(* IEC 61131-3 sources: std_i2980_v2.06_cp053/Source/IMM/ieccontrol/OperationMode1 (part 3) *)

(* ---- ABProduction.pu ---- *)
(*
@h    ! WARNING !
@h    The Kemro K2 system (including software) only meets category B according to EN 954-1,
@h    thus it is not intended for usage in safety-relevant control applications in the field
@h    of personal safety (e.g. emergency stop).
@h    To implement potentially necessary safety-relevant control tasks, always use additional
@h    external safety devices that are intended for the particular purpose, and meet the necessary
@h    functional safety.
@h    For further information see EN 954-1 (EN ISO 13849-1) and/or the K2-x00 user manual, chapter
@h    "CE conformity, directives and standards".

production statistic (good/bad part)
called by ABShotCounter in order to provide some additional production information
*)

IMPORT_OVER_LISTFILE
 cCompPDP
, cCompMotionProtectMold
, tsTraceLevel
, tevPartCheck
, tnBadPartReason
, tsProduction
, RTC
, FBDebugTrace
, tevPartCheckData

END_IMPORT

ALGORITHM_BLOCK ABProduction #DUMMY_EDIT_BLOCK

SYSTEM_VAR
 sv_TraceLevel : tsTraceLevel;
 sv_bBadPart : BOOL;
 sv_iProdCounterAct : DINT;
 sv_iShotCounterRetain : UDINT (* shot counter retain (used for lubrication) *);
 sv_iCavities : DINT;
 sv_BadPartReason : tnBadPartReason;
 sv_Production : tsProduction;
 sv_dShotTimeAct : DATE_AND_TIME;
END_VAR

SYSTEM_OBJECT
 evPartCheck : tevPartCheck;
 EV_Task_7 : TASK;
 PU_Task_7 : TASK;
END_OBJECT

VAR
 miRejectsPerTime : DINT;
 fbRtc : RTC;
 mdStartTime : DT;
 fbDebugTrace : FBDebugTrace;
END_VAR

(*
@h    ! WARNING !
@h    The Kemro K2 system (including software) only meets category B according to EN 954-1,
@h    thus it is not intended for usage in safety-relevant control applications in the field
@h    of personal safety (e.g. emergency stop).
@h    To implement potentially necessary safety-relevant control tasks, always use additional
@h    external safety devices that are intended for the particular purpose, and meet the necessary
@h    functional safety.
@h    For further information see EN 954-1 (EN ISO 13849-1) and/or the K2-x00 user manual, chapter
@h    "CE conformity, directives and standards".

reacts on partcheck events with bBadPart == TRUE,
sets sv_bBadPart and sv_BadPartReason
*)

EVENT_ALGORITHM evaPartCheck ON EV_Task_7 WITH evPartCheck

VAR_INPUT
 partCheckData : tevPartCheckData;
END_VAR

VAR
 s : STRING(255);
END_VAR
#BEGIN_EDIT_BLOCK
(**************************************** WARNING ********************************************
 *** The KEBA Kemro K2 System including software is not intended for safety control tasks! ***
 ***                       For further information see Comment tab!                        ***
 *********************************************************************************************)

IF sv_TraceLevel.bApplication THEN
    s := CONCAT('part check event recieved: device ',
                DINT_TO_STRING(partCheckData.DeviceID.CompId),
                '/',
                DINT_TO_STRING(partCheckData.DeviceID.IndexId),
                ' bad ',
                BOOL_TO_STRING(partCheckData.bBadPart),
                ' reject',
                BOOL_TO_STRING(partCheckData.bReject)
            );
    fbDebugTrace(sText := s);
END_IF;

IF partCheckData.bBadPart THEN
    sv_bBadPart := TRUE;

    // set bad part reason
    IF sv_BadPartReason = nReason_GoodPart THEN
       CASE (partCheckData.DeviceID.CompId) OF
            cCompPDP:
                 sv_BadPartReason := nReason_PDS;

            cCompMotionProtectMold:
                 sv_BadPartReason := nReason_MoldProtection;
       ELSE
             sv_BadPartReason := nReason_Unknown;
       END_CASE;
    END_IF;

END_IF;

;#END_EDIT_BLOCK END_ALGORITHM

(*
@h    ! WARNING !
@h    The Kemro K2 system (including software) only meets category B according to EN 954-1,
@h    thus it is not intended for usage in safety-relevant control applications in the field
@h    of personal safety (e.g. emergency stop).
@h    To implement potentially necessary safety-relevant control tasks, always use additional
@h    external safety devices that are intended for the particular purpose, and meet the necessary
@h    functional safety.
@h    For further information see EN 954-1 (EN ISO 13849-1) and/or the K2-x00 user manual, chapter
@h    "CE conformity, directives and standards".

called by ABShotCounter before shotcounter is increased, so sv_Production vars that can be recorded
by PDP are written before sampled by PDP
*)

ALGORITHM aNewCycle

#BEGIN_EDIT_BLOCK
(**************************************** WARNING ********************************************
 *** The KEBA Kemro K2 System including software is not intended for safety control tasks! ***
 ***                       For further information see Comment tab!                        ***
 *********************************************************************************************)

// end of actual cycle, calc some production data

fbRtc();
sv_dShotTimeAct := fbRtc.CDT;

IF ((fbRtc.CDT - mdStartTime) >= LINT_TO_TIME(DINT_TO_LINT(sv_Production.iRejectTimeSpan * 60 * 1000) * 1000)) THEN
    mdStartTime := fbRtc.CDT;
    sv_Production.iRejectsPerTime := miRejectsPerTime;
    miRejectsPerTime := 0;
END_IF;

IF sv_bBadPart THEN
    sv_Production.iRejectCounter := sv_Production.iRejectCounter + sv_iCavities;
    miRejectsPerTime := miRejectsPerTime + sv_iCavities;
    sv_Production.iRejectsInSeries := sv_Production.iRejectsInSeries + 1;
ELSE
    sv_Production.iRejectsInSeries := 0;
END_IF;

IF sv_Production.iRejectCounter > 0 THEN
    sv_Production.iGoodPartsPerReject := (sv_iProdCounterAct - sv_Production.iRejectCounter) / sv_Production.iRejectCounter;
END_IF;

;#END_EDIT_BLOCK END_ALGORITHM

(*
@h    ! WARNING !
@h    The Kemro K2 system (including software) only meets category B according to EN 954-1,
@h    thus it is not intended for usage in safety-relevant control applications in the field
@h    of personal safety (e.g. emergency stop).
@h    To implement potentially necessary safety-relevant control tasks, always use additional
@h    external safety devices that are intended for the particular purpose, and meet the necessary
@h    functional safety.
@h    For further information see EN 954-1 (EN ISO 13849-1) and/or the K2-x00 user manual, chapter
@h    "CE conformity, directives and standards".

called by ABShotCounter when shotcounter is reset
to clear all production statistics variables also
*)

ALGORITHM aResetData

#BEGIN_EDIT_BLOCK
(**************************************** WARNING ********************************************
 *** The KEBA Kemro K2 System including software is not intended for safety control tasks! ***
 ***                       For further information see Comment tab!                        ***
 *********************************************************************************************)

sv_Production.iRejectCounter := 0;
sv_Production.iRejectsPerTime := 0;
sv_Production.iGoodPartsPerReject := 2147483647;
sv_Production.iRejectsInSeries := 0;

miRejectsPerTime := 0;
fbRtc();
mdStartTime := fbRtc.CDT;

;#END_EDIT_BLOCK END_ALGORITHM

(*
@h    ! WARNING !
@h    The Kemro K2 system (including software) only meets category B according to EN 954-1,
@h    thus it is not intended for usage in safety-relevant control applications in the field
@h    of personal safety (e.g. emergency stop).
@h    To implement potentially necessary safety-relevant control tasks, always use additional
@h    external safety devices that are intended for the particular purpose, and meet the necessary
@h    functional safety.
@h    For further information see EN 954-1 (EN ISO 13849-1) and/or the K2-x00 user manual, chapter
@h    "CE conformity, directives and standards".

called when new cycle starts (shotcounter has just been increased) but lower prio than PDP recording
so SVs to be recorded by PDP are sampled before reset
*)

POSTUPDATE_ALGORITHM pNewCycle ON PU_Task_7 WITH sv_iShotCounterRetain

#BEGIN_EDIT_BLOCK
(**************************************** WARNING ********************************************
 *** The KEBA Kemro K2 System including software is not intended for safety control tasks! ***
 ***                       For further information see Comment tab!                        ***
 *********************************************************************************************)

//reset bad part
// ATTENTION: lower prio than PDP MS Task so PDP has recorded these SVs before reset!

sv_bBadPart := FALSE;
sv_BadPartReason := nReason_GoodPart;

;#END_EDIT_BLOCK END_ALGORITHM

END_ALGORITHM_BLOCK

#END_OF_IEC_PART

@Puma @IecEditor 6 103 @Pou 25
@@@BEG_Comment@@@
@h    ! WARNING !
@h    The Kemro K2 system (including software) only meets category B according to EN 954-1,
@h    thus it is not intended for usage in safety-relevant control applications in the field
@h    of personal safety (e.g. emergency stop).
@h    To implement potentially necessary safety-relevant control tasks, always use additional
@h    external safety devices that are intended for the particular purpose, and meet the necessary
@h    functional safety.
@h    For further information see EN 954-1 (EN ISO 13849-1) and/or the K2-x00 user manual, chapter
@h    "CE conformity, directives and standards".

production statistic (good/bad part)
called by ABShotCounter in order to provide some additional production information
@@@END_Comment@@@

@BEG_Contents

@BEG_Func
@RT(17)FuncTreeContainer
0
@END_Func

@BEG_Const
@RT(18)ConstTreeContainer
2
@Var @RT(8)cCompPDP @RT(0) @T @F @DT @RT(4)DINT @RT(0) @T @T @BASIC 0 @F
@F @F
@T
@BEG_Attrib
0 @RT(3)119 @RT(30)Component Process Data Package
@END_Attrib
1 1 @F @F @F @F

@Var @RT(22)cCompMotionProtectMold @RT(0) @T @F @DT @RT(4)DINT @RT(0) @T @T @BASIC 0 @F
@F @F
@T
@BEG_Attrib
0 @RT(3)130 @RT(29)Component Motion Protect Mold
@END_Attrib
1 1 @F @F @F @F

@END_Const

@BEG_Export

@BEG_Kind
@ALGORITHM_BLOCK @RT(12)ABProduction @STRUCTURED_TEXT
@RT(0) @RT(0) @RT(0)
@END_Kind

@BEG_Dcl
@RT(16)DclTreeContainer
15
@Var @RT(13)sv_TraceLevel @RT(0) @T @T @DERIVED 0 @T @T @DT @RT(12)tsTraceLevel @RT(0) @T @T @UNKNOWN 0 @F
@F @F
@T
@BEG_Attrib
3 @RT(0) @RT(0) @RT(0)
@END_Attrib
1 8 @F @F @F @F

@Var @RT(11)evPartCheck @RT(0) @T @T @DERIVED 0 @T @T @DT @RT(12)tevPartCheck @RT(0) @T @T @UNKNOWN 0 @F
@F @F
@T
@BEG_Attrib
3 @RT(0) @RT(0) @RT(0)
@END_Attrib
1 7 @F @F @F @F

@Var @RT(9)EV_Task_7 @RT(0) @T @T @RENAMED 0 @T @T @DT @RT(4)TASK @RT(0) @T @T @BASIC 0 @F
@F @F
@T
@BEG_Attrib
3 @RT(0) @RT(0) @RT(0)
@END_Attrib
1 7 @F @F @F @F

@Var @RT(11)sv_bBadPart @RT(0) @T @F @DT @RT(4)BOOL @RT(0) @T @T @BASIC 0 @F
@F @F
@T
@BEG_Attrib
3 @RT(0) @RT(0) @RT(0)
@END_Attrib
1 8 @F @F @F @F

@Var @RT(18)sv_iProdCounterAct @RT(0) @T @F @DT @RT(4)DINT @RT(0) @T @T @BASIC 0 @F
@F @F
@T
@BEG_Attrib
3 @RT(0) @RT(0) @RT(0)
@END_Attrib
1 8 @F @F @F @F

@Var @RT(21)sv_iShotCounterRetain @RT(0) @T @F @DT @RT(5)UDINT @RT(0) @T @T @BASIC 0 @F
@F @F
@T
@BEG_Attrib
3 @RT(0) @RT(42)shot counter retain (used for lubrication) @RT(0)
@END_Attrib
1 8 @F @F @F @F

@Var @RT(12)sv_iCavities @RT(0) @T @F @DT @RT(4)DINT @RT(0) @T @T @BASIC 0 @F
@F @F
@T
@BEG_Attrib
3 @RT(0) @RT(0) @RT(0)
@END_Attrib
1 8 @F @F @F @F

@Var @RT(16)sv_BadPartReason @RT(0) @T @T @DERIVED 0 @T @T @DT @RT(15)tnBadPartReason @RT(0) @T @T @UNKNOWN 0 @F
@F @F
@T
@BEG_Attrib
3 @RT(0) @RT(0) @RT(0)
@END_Attrib
1 8 @F @F @F @F

@Var @RT(13)sv_Production @RT(0) @T @T @DERIVED 0 @T @T @DT @RT(12)tsProduction @RT(0) @T @T @UNKNOWN 0 @F
@F @F
@T
@BEG_Attrib
3 @RT(0) @RT(0) @RT(0)
@END_Attrib
1 8 @F @F @F @F

@Var @RT(16)miRejectsPerTime @RT(0) @T @F @DT @RT(4)DINT @RT(0) @T @T @BASIC 0 @F
@F @F
@T
@BEG_Attrib
3 @RT(0) @RT(0) @RT(0)
@END_Attrib
1 0 @F @F @F @F

@Var @RT(5)fbRtc @RT(0) @T @T @DERIVED 0 @T @T @DT @RT(3)RTC @RT(0) @T @T @UNKNOWN 0 @F
@F @F
@T
@BEG_Attrib
3 @RT(0) @RT(0) @RT(0)
@END_Attrib
1 0 @F @F @F @F

@Var @RT(15)sv_dShotTimeAct @RT(0) @T @F @DT @RT(13)DATE_AND_TIME @RT(0) @T @T @BASIC 0 @F
@F @F
@T
@BEG_Attrib
3 @RT(0) @RT(0) @RT(0)
@END_Attrib
1 8 @F @F @F @F

@Var @RT(11)mdStartTime @RT(0) @T @F @DT @RT(2)DT @RT(0) @T @T @BASIC 0 @F
@F @F
@T
@BEG_Attrib
3 @RT(0) @RT(0) @RT(0)
@END_Attrib
1 0 @F @F @F @F

@Var @RT(9)PU_Task_7 @RT(0) @T @T @RENAMED 0 @T @T @DT @RT(4)TASK @RT(0) @T @T @BASIC 0 @F
@F @F
@T
@BEG_Attrib
3 @RT(0) @RT(0) @RT(0)
@END_Attrib
1 7 @F @F @F @F

@Var @RT(12)fbDebugTrace @RT(0) @T @T @DERIVED 0 @T @T @DT @RT(12)FBDebugTrace @RT(0) @T @T @UNKNOWN 0 @F
@F @F
@T
@BEG_Attrib
3 @RT(0) @RT(0) @RT(0)
@END_Attrib
1 0 @F @F @F @F

@END_Dcl

@END_Export

@BEG_Body

4

@BEG_Export

@BEG_Algo
@EVENT_ALGORITHM @RT(12)evaPartCheck @STRUCTURED_TEXT
@RT(0) @RT(11)evPartCheck @RT(9)EV_Task_7 @F @F
@END_Algo

@BEG_Dcl
@RT(16)DclTreeContainer
2
@Var @RT(13)partCheckData @RT(0) @T @T @DERIVED 0 @T @T @DT @RT(16)tevPartCheckData @RT(0) @T @T @UNKNOWN 0 @F
@F @F
@T
@BEG_Attrib
3 @RT(0) @RT(0) @RT(0)
@END_Attrib
1 1 @F @F @F @F

@Var @RT(1)s @RT(0) @T @F @DT @RT(11)STRING(255) @RT(0) @T @T @STRING 0 @F @RT(3)255 @F
@F @F
@T
@BEG_Attrib
3 @RT(0) @RT(0) @RT(0)
@END_Attrib
1 0 @F @F @F @F

@END_Dcl

@END_Export

@BEG_Export

@BEG_Algo
@ALGORITHM @RT(9)aNewCycle @STRUCTURED_TEXT
@RT(0) @RT(0) @RT(0) @F @F
@END_Algo

@BEG_Dcl
@RT(16)DclTreeContainer
0
@END_Dcl

@END_Export

@BEG_Export

@BEG_Algo
@ALGORITHM @RT(10)aResetData @STRUCTURED_TEXT
@RT(0) @RT(0) @RT(0) @F @F
@END_Algo

@BEG_Dcl
@RT(16)DclTreeContainer
0
@END_Dcl

@END_Export

@BEG_Export

@BEG_Algo
@POSTUPDATE_ALGORITHM @RT(9)pNewCycle @STRUCTURED_TEXT
@RT(0) @RT(21)sv_iShotCounterRetain @RT(9)PU_Task_7 @F @F
@END_Algo

@BEG_Dcl
@RT(16)DclTreeContainer
0
@END_Dcl

@END_Export

@BEG_Body
@TL(38)
(**************************************** WARNING ********************************************
 *** The KEBA Kemro K2 System including software is not intended for safety control tasks! ***
 ***                       For further information see Comment tab!                        ***
 *********************************************************************************************)

IF sv_TraceLevel.bApplication THEN
    s := CONCAT('part check event recieved: device ',
                DINT_TO_STRING(partCheckData.DeviceID.CompId),
                '/',
                DINT_TO_STRING(partCheckData.DeviceID.IndexId),
                ' bad ',
                BOOL_TO_STRING(partCheckData.bBadPart),
                ' reject',
                BOOL_TO_STRING(partCheckData.bReject)
            );
    fbDebugTrace(sText := s);
END_IF;

IF partCheckData.bBadPart THEN
    sv_bBadPart := TRUE;

    // set bad part reason
    IF sv_BadPartReason = nReason_GoodPart THEN
       CASE (partCheckData.DeviceID.CompId) OF
            cCompPDP:
                 sv_BadPartReason := nReason_PDS;

            cCompMotionProtectMold:
                 sv_BadPartReason := nReason_MoldProtection;
       ELSE
             sv_BadPartReason := nReason_Unknown;
       END_CASE;
    END_IF;

END_IF;

@END_Body

@@@BEG_Comment@@@
@TL(12)
@h    ! WARNING !
@h    The Kemro K2 system (including software) only meets category B according to EN 954-1,
@h    thus it is not intended for usage in safety-relevant control applications in the field
@h    of personal safety (e.g. emergency stop).
@h    To implement potentially necessary safety-relevant control tasks, always use additional
@h    external safety devices that are intended for the particular purpose, and meet the necessary
@h    functional safety.
@h    For further information see EN 954-1 (EN ISO 13849-1) and/or the K2-x00 user manual, chapter
@h    "CE conformity, directives and standards".

reacts on partcheck events with bBadPart == TRUE,
sets sv_bBadPart and sv_BadPartReason
@@@END_Comment@@@

@BEG_Body
@TL(30)
(**************************************** WARNING ********************************************
 *** The KEBA Kemro K2 System including software is not intended for safety control tasks! ***
 ***                       For further information see Comment tab!                        ***
 *********************************************************************************************)

// end of actual cycle, calc some production data

fbRtc();
sv_dShotTimeAct := fbRtc.CDT;

IF ((fbRtc.CDT - mdStartTime) >= LINT_TO_TIME(DINT_TO_LINT(sv_Production.iRejectTimeSpan * 60 * 1000) * 1000)) THEN
    mdStartTime := fbRtc.CDT;
    sv_Production.iRejectsPerTime := miRejectsPerTime;
    miRejectsPerTime := 0;
END_IF;

IF sv_bBadPart THEN
    sv_Production.iRejectCounter := sv_Production.iRejectCounter + sv_iCavities;
    miRejectsPerTime := miRejectsPerTime + sv_iCavities;
    sv_Production.iRejectsInSeries := sv_Production.iRejectsInSeries + 1;
ELSE
    sv_Production.iRejectsInSeries := 0;
END_IF;

IF sv_Production.iRejectCounter > 0 THEN
    sv_Production.iGoodPartsPerReject := (sv_iProdCounterAct - sv_Production.iRejectCounter) / sv_Production.iRejectCounter;
END_IF;

@END_Body

@@@BEG_Comment@@@
@TL(12)
@h    ! WARNING !
@h    The Kemro K2 system (including software) only meets category B according to EN 954-1,
@h    thus it is not intended for usage in safety-relevant control applications in the field
@h    of personal safety (e.g. emergency stop).
@h    To implement potentially necessary safety-relevant control tasks, always use additional
@h    external safety devices that are intended for the particular purpose, and meet the necessary
@h    functional safety.
@h    For further information see EN 954-1 (EN ISO 13849-1) and/or the K2-x00 user manual, chapter
@h    "CE conformity, directives and standards".

called by ABShotCounter before shotcounter is increased, so sv_Production vars that can be recorded
by PDP are written before sampled by PDP
@@@END_Comment@@@

@BEG_Body
@TL(14)
(**************************************** WARNING ********************************************
 *** The KEBA Kemro K2 System including software is not intended for safety control tasks! ***
 ***                       For further information see Comment tab!                        ***
 *********************************************************************************************)

sv_Production.iRejectCounter := 0;
sv_Production.iRejectsPerTime := 0;
sv_Production.iGoodPartsPerReject := 2147483647;
sv_Production.iRejectsInSeries := 0;

miRejectsPerTime := 0;
fbRtc();
mdStartTime := fbRtc.CDT;

@END_Body

@@@BEG_Comment@@@
@TL(12)
@h    ! WARNING !
@h    The Kemro K2 system (including software) only meets category B according to EN 954-1,
@h    thus it is not intended for usage in safety-relevant control applications in the field
@h    of personal safety (e.g. emergency stop).
@h    To implement potentially necessary safety-relevant control tasks, always use additional
@h    external safety devices that are intended for the particular purpose, and meet the necessary
@h    functional safety.
@h    For further information see EN 954-1 (EN ISO 13849-1) and/or the K2-x00 user manual, chapter
@h    "CE conformity, directives and standards".

called by ABShotCounter when shotcounter is reset
to clear all production statistics variables also
@@@END_Comment@@@

@BEG_Body
@TL(12)
(**************************************** WARNING ********************************************
 *** The KEBA Kemro K2 System including software is not intended for safety control tasks! ***
 ***                       For further information see Comment tab!                        ***
 *********************************************************************************************)

//reset bad part
// ATTENTION: lower prio than PDP MS Task so PDP has recorded these SVs before reset!

sv_bBadPart := FALSE;
sv_BadPartReason := nReason_GoodPart;

@END_Body

@@@BEG_Comment@@@
@TL(12)
@h    ! WARNING !
@h    The Kemro K2 system (including software) only meets category B according to EN 954-1,
@h    thus it is not intended for usage in safety-relevant control applications in the field
@h    of personal safety (e.g. emergency stop).
@h    To implement potentially necessary safety-relevant control tasks, always use additional
@h    external safety devices that are intended for the particular purpose, and meet the necessary
@h    functional safety.
@h    For further information see EN 954-1 (EN ISO 13849-1) and/or the K2-x00 user manual, chapter
@h    "CE conformity, directives and standards".

called when new cycle starts (shotcounter has just been increased) but lower prio than PDP recording
so SVs to be recorded by PDP are sampled before reset
@@@END_Comment@@@
@END_Body

@END_Contents

(* ---- ABSequenceInterruption.pu ---- *)
(*
@h    ! WARNING !
@h    The Kemro K2 system (including software) only meets category B according to EN 954-1,
@h    thus it is not intended for usage in safety-relevant control applications in the field
@h    of personal safety (e.g. emergency stop).
@h    To implement potentially necessary safety-relevant control tasks, always use additional
@h    external safety devices that are intended for the particular purpose, and meet the necessary
@h    functional safety.
@h    For further information see EN 954-1 (EN ISO 13849-1) and/or the K2-x00 user manual, chapter
@h    "CE conformity, directives and standards".

This AB is responsible for setting / resetting the flag for sequence interruption (sv_bSequenceInterruption).
A sequence interruption can be triggered by any function unit. Therefore and according event (evSequenceInterrupt)
must be sent.
This block can also handle a seperate digital input (di_SequenceInterruption) which can trigger an interrupt.
Interrupt events (or the according digital input) are ignored in manual and setup mode.

During sequence is interrupted, the led for halfautocycle or fullautocycle is set to "flashing"

*)

IMPORT_OVER_LISTFILE
 tnOperationMode
, tevSequenceInterrupt
, tsActiveMovements
, tevSequInterruptData

END_IMPORT

ALGORITHM_BLOCK ABSequenceInterruption #DUMMY_EDIT_BLOCK

SYSTEM_VAR
 di_SequenceInterruption : BOOL;
 sv_bSequenceInterruption : BOOL (* TRUE: sequence is interrupted *);
 sv_bLedHalfAutomatic_ledAttr : BYTE (* Panel LED half automatic *);
 sv_bLedFullAutomatic_ledAttr : BYTE (* Panel LED full automatic *);
 sv_bHMILedHalfAutomatic_ledAttr : BYTE (* Panel LED half automatic *);
 sv_bHMILedFullAutomatic_ledAttr : BYTE (* Panel LED full automatic *);
 sv_OperationMode : tnOperationMode;
 sv_ActiveMovements : tsActiveMovements;
END_VAR

SYSTEM_OBJECT
 PU_Task_7 : TASK;
 EV_Task_7 : TASK;
 evSequenceInterrupt : tevSequenceInterrupt;
 TaskMid : TASK;
END_OBJECT

VAR
 mbLedHalfAutomaticAttrLinked : BOOL;
 mbLedFullAutomaticAttrLinked : BOOL;
 mbResetInterrupt : BOOL;
END_VAR

POSTUPDATE_ALGORITHM pDISequenceInterrupt ON PU_Task_7 WITH di_SequenceInterruption

VAR
 evSequenceInterruptData : tevSequInterruptData;
END_VAR
#BEGIN_EDIT_BLOCK
(**************************************** WARNING ********************************************
 *** The KEBA Kemro K2 System including software is not intended for safety control tasks! ***
 ***                       For further information see Comment tab!                        ***
 *********************************************************************************************)

IF di_SequenceInterruption THEN
   IF sv_bSequenceInterruption THEN
      evSequenceInterruptData.SequenceInterrupt := nSequenceContinue;
   ELSE
      evSequenceInterruptData.SequenceInterrupt := nSequenceInterrupt;
   END_IF;

   SET_EVENT(evSequenceInterrupt, evSequenceInterruptData);
END_IF;

;#END_EDIT_BLOCK END_ALGORITHM

EVENT_ALGORITHM evaSequenceInterrupt ON EV_Task_7 WITH evSequenceInterrupt

VAR_INPUT
 evSequInterruptData : tevSequInterruptData;
END_VAR
#BEGIN_EDIT_BLOCK
(**************************************** WARNING ********************************************
 *** The KEBA Kemro K2 System including software is not intended for safety control tasks! ***
 ***                       For further information see Comment tab!                        ***
 *********************************************************************************************)

IF (sv_OperationMode = nSetup) OR (sv_OperationMode = nManual) THEN
   RETURN;
END_IF;

IF evSequInterruptData.SequenceInterrupt = nSequenceInterrupt THEN
   sv_bSequenceInterruption := TRUE;
   mbResetInterrupt := FALSE;

   //set led attribute to "flashing" during sequence interrupt
   sv_bLedHalfAutomatic_ledAttr := 16#3;
   sv_bLedFullAutomatic_ledAttr := 16#3;

   sv_bHMILedHalfAutomatic_ledAttr := sv_bLedHalfAutomatic_ledAttr;
   sv_bHMILedFullAutomatic_ledAttr := sv_bLedFullAutomatic_ledAttr;

   START_PROCESS_ALGORITHM(paSequenceInterrupted);
ELSE
   mbResetInterrupt := TRUE;
END_IF;

;#END_EDIT_BLOCK END_ALGORITHM

PROCESS_ALGORITHM paSequenceInterrupted ON TaskMid

(* IecGraph-Code *)

(* init step *)
INITIAL_STEP S_Init:
Action9 (P);
END_STEP

ACTION Action9: #BEGIN_EDIT_BLOCK

mbLedHalfAutomaticAttrLinked := IS_LINKED(sv_bLedHalfAutomatic_ledAttr);
mbLedFullAutomaticAttrLinked := IS_LINKED(sv_bLedFullAutomatic_ledAttr);

;#END_EDIT_BLOCK END_ACTION (*Action9*)

(* steps *)
STEP S_Interrupted:
END_STEP

STEP S_WaitNoMove:
END_STEP

STEP S_Stop:
AReset (P);
AStop (P);
END_STEP

ACTION AReset: #BEGIN_EDIT_BLOCK
sv_bSequenceInterruption := FALSE;
//set led attribute to "not flashing"
sv_bHMILedHalfAutomatic_ledAttr := 16#1;
sv_bHMILedFullAutomatic_ledAttr := 16#1;

IF mbLedHalfAutomaticAttrLinked THEN
   sv_bLedHalfAutomatic_ledAttr := sv_bHMILedHalfAutomatic_ledAttr;
END_IF;

IF mbLedFullAutomaticAttrLinked THEN
   sv_bLedFullAutomatic_ledAttr := sv_bHMILedFullAutomatic_ledAttr;
END_IF;

;#END_EDIT_BLOCK END_ACTION (*AReset*)
ACTION AStop: #BEGIN_EDIT_BLOCK
STOP_PROCESS_ALGORITHM();

;#END_EDIT_BLOCK END_ACTION (*AStop*)

(* transitions *)
GO_ON_TRANSITION Trans1 (* Trans1 *) FROM S_Init TO S_Interrupted :=  #BEGIN_EDIT_BLOCK
TRUE
;#END_EDIT_BLOCK
END_TRANSITION

GO_ON_TRANSITION TResetInterrupt (* Trans2 *) FROM S_Interrupted TO S_WaitNoMove :=  #BEGIN_EDIT_BLOCK
mbResetInterrupt
;#END_EDIT_BLOCK
END_TRANSITION

GO_ON_TRANSITION TNoMovementActive (* Trans4 *) FROM S_WaitNoMove TO S_Stop :=  #BEGIN_EDIT_BLOCK
sv_ActiveMovements.iNumberOfActiveMovements = 0
;#END_EDIT_BLOCK
END_TRANSITION

GO_ON_TRANSITION TOpModeChanged (* Trans8 *) FROM S_Interrupted TO S_Stop :=  #BEGIN_EDIT_BLOCK
sv_OperationMode < nHalfAutomatic
;#END_EDIT_BLOCK
END_TRANSITION

TRANSITION Trans3 (* Trans3 *) FROM S_Stop TO S_Interrupted :=  #BEGIN_EDIT_BLOCK
TRUE
;#END_EDIT_BLOCK
END_TRANSITION

(* end IecGraph-Code *)
(* sfc-code *)

(* stand alone actions *)
// ACTION Action9: #BEGIN_EDIT_BLOCK

// ;#END_EDIT_BLOCK END_ACTION (*Action9*)
(* end sfc-code *)

END_ALGORITHM

END_ALGORITHM_BLOCK

#END_OF_IEC_PART

@Puma @IecEditor 6 131 @Pou 25
@@@BEG_Comment@@@
@h    ! WARNING !
@h    The Kemro K2 system (including software) only meets category B according to EN 954-1,
@h    thus it is not intended for usage in safety-relevant control applications in the field
@h    of personal safety (e.g. emergency stop).
@h    To implement potentially necessary safety-relevant control tasks, always use additional
@h    external safety devices that are intended for the particular purpose, and meet the necessary
@h    functional safety.
@h    For further information see EN 954-1 (EN ISO 13849-1) and/or the K2-x00 user manual, chapter
@h    "CE conformity, directives and standards".

This AB is responsible for setting / resetting the flag for sequence interruption (sv_bSequenceInterruption).
A sequence interruption can be triggered by any function unit. Therefore and according event (evSequenceInterrupt)
must be sent.
This block can also handle a seperate digital input (di_SequenceInterruption) which can trigger an interrupt.
Interrupt events (or the according digital input) are ignored in manual and setup mode.

During sequence is interrupted, the led for halfautocycle or fullautocycle is set to "flashing"

@@@END_Comment@@@

@BEG_Contents

@BEG_Func
@RT(17)FuncTreeContainer
0
@END_Func

@BEG_Const
@RT(18)ConstTreeContainer
0
@END_Const

@BEG_Export

@BEG_Kind
@ALGORITHM_BLOCK @RT(22)ABSequenceInterruption @STRUCTURED_TEXT
@RT(0) @RT(0) @RT(0)
@END_Kind

@BEG_Dcl
@RT(16)DclTreeContainer
15
@Var @RT(23)di_SequenceInterruption @RT(0) @T @F @DT @RT(4)BOOL @RT(0) @T @T @BASIC 0 @F
@F @F
@T
@BEG_Attrib
3 @RT(0) @RT(0) @RT(0)
@END_Attrib
1 8 @F @F @F @F

@Var @RT(9)PU_Task_7 @RT(0) @T @T @RENAMED 0 @T @T @DT @RT(4)TASK @RT(0) @T @T @BASIC 0 @F
@F @F
@T
@BEG_Attrib
3 @RT(0) @RT(0) @RT(0)
@END_Attrib
1 7 @F @F @F @F

@Var @RT(24)sv_bSequenceInterruption @RT(0) @T @F @DT @RT(4)BOOL @RT(0) @T @T @BASIC 0 @F
@F @F
@T
@BEG_Attrib
3 @RT(0) @RT(29)TRUE: sequence is interrupted @RT(0)
@END_Attrib
1 8 @F @F @F @F

@Var @RT(28)sv_bLedHalfAutomatic_ledAttr @RT(0) @T @F @DT @RT(4)BYTE @RT(0) @T @T @BASIC 0 @F
@F @F
@T
@BEG_Attrib
3 @RT(0) @RT(24)Panel LED half automatic @RT(0)
@END_Attrib
1 8 @F @F @F @F

@Var @RT(28)sv_bLedFullAutomatic_ledAttr @RT(0) @T @F @DT @RT(4)BYTE @RT(0) @T @T @BASIC 0 @F
@F @F
@T
@BEG_Attrib
3 @RT(0) @RT(24)Panel LED full automatic @RT(0)
@END_Attrib
1 8 @F @F @F @F

@Var @RT(31)sv_bHMILedHalfAutomatic_ledAttr @RT(0) @T @F @DT @RT(4)BYTE @RT(0) @T @T @BASIC 0 @F
@F @F
@T
@BEG_Attrib
3 @RT(0) @RT(24)Panel LED half automatic @RT(0)
@END_Attrib
1 8 @F @F @F @F

@Var @RT(31)sv_bHMILedFullAutomatic_ledAttr @RT(0) @T @F @DT @RT(4)BYTE @RT(0) @T @T @BASIC 0 @F
@F @F
@T
@BEG_Attrib
3 @RT(0) @RT(24)Panel LED full automatic @RT(0)
@END_Attrib
1 8 @F @F @F @F

@Var @RT(16)sv_OperationMode @RT(0) @T @T @DERIVED 0 @T @T @DT @RT(15)tnOperationMode @RT(0) @T @T @UNKNOWN 0 @F
@F @F
@T
@BEG_Attrib
3 @RT(0) @RT(0) @RT(0)
@END_Attrib
1 8 @F @F @F @F

@Var @RT(9)EV_Task_7 @RT(0) @T @T @RENAMED 0 @T @T @DT @RT(4)TASK @RT(0) @T @T @BASIC 0 @F
@F @F
@T
@BEG_Attrib
3 @RT(0) @RT(0) @RT(0)
@END_Attrib
1 7 @F @F @F @F

@Var @RT(19)evSequenceInterrupt @RT(0) @T @T @DERIVED 0 @T @T @DT @RT(20)tevSequenceInterrupt @RT(0) @T @T @UNKNOWN 0 @F
@F @F
@T
@BEG_Attrib
3 @RT(0) @RT(0) @RT(0)
@END_Attrib
1 7 @F @F @F @F

@Var @RT(7)TaskMid @RT(0) @T @T @RENAMED 0 @T @T @DT @RT(4)TASK @RT(0) @T @T @BASIC 0 @F
@F @F
@T
@BEG_Attrib
3 @RT(0) @RT(0) @RT(0)
@END_Attrib
1 7 @F @F @F @F

@Var @RT(28)mbLedHalfAutomaticAttrLinked @RT(0) @T @F @DT @RT(4)BOOL @RT(0) @T @T @BASIC 0 @F
@F @F
@T
@BEG_Attrib
3 @RT(0) @RT(0) @RT(0)
@END_Attrib
1 0 @F @F @F @F

@Var @RT(28)mbLedFullAutomaticAttrLinked @RT(0) @T @F @DT @RT(4)BOOL @RT(0) @T @T @BASIC 0 @F
@F @F
@T
@BEG_Attrib
3 @RT(0) @RT(0) @RT(0)
@END_Attrib
1 0 @F @F @F @F

@Var @RT(16)mbResetInterrupt @RT(0) @T @F @DT @RT(4)BOOL @RT(0) @T @T @BASIC 0 @F
@F @F
@T
@BEG_Attrib
3 @RT(0) @RT(0) @RT(0)
@END_Attrib
1 0 @F @F @F @F

@Var @RT(18)sv_ActiveMovements @RT(0) @T @T @DERIVED 0 @T @T @DT @RT(17)tsActiveMovements @RT(0) @T @T @UNKNOWN 0 @F
@F @F
@T
@BEG_Attrib
3 @RT(0) @RT(0) @RT(0)
@END_Attrib
1 8 @F @F @F @F

@END_Dcl

@END_Export

@BEG_Body

3

@BEG_Export

@BEG_Algo
@POSTUPDATE_ALGORITHM @RT(20)pDISequenceInterrupt @STRUCTURED_TEXT
@RT(0) @RT(23)di_SequenceInterruption @RT(9)PU_Task_7 @F @F
@END_Algo

@BEG_Dcl
@RT(16)DclTreeContainer
1
@Var @RT(23)evSequenceInterruptData @RT(0) @T @T @DERIVED 0 @T @T @DT @RT(20)tevSequInterruptData @RT(0) @T @T @UNKNOWN 0 @F
@F @F
@T
@BEG_Attrib
3 @RT(0) @RT(0) @RT(0)
@END_Attrib
1 0 @F @F @F @F

@END_Dcl

@END_Export

@BEG_Export

@BEG_Algo
@EVENT_ALGORITHM @RT(20)evaSequenceInterrupt @STRUCTURED_TEXT
@RT(0) @RT(19)evSequenceInterrupt @RT(9)EV_Task_7 @F @F
@END_Algo

@BEG_Dcl
@RT(16)DclTreeContainer
1
@Var @RT(19)evSequInterruptData @RT(0) @T @T @DERIVED 0 @T @T @DT @RT(20)tevSequInterruptData @RT(0) @T @T @UNKNOWN 0 @F
@F @F
@T
@BEG_Attrib
3 @RT(0) @RT(0) @RT(0)
@END_Attrib
1 1 @F @F @F @F

@END_Dcl

@END_Export

@BEG_Export

@BEG_Algo
@PROCESS_ALGORITHM @RT(21)paSequenceInterrupted @SEQUENTIAL_FLOW_CHART
@RT(0) @RT(0) @RT(7)TaskMid @F @F
@END_Algo

@BEG_Dcl
@RT(16)DclTreeContainer
0
@END_Dcl

@END_Export

@BEG_Body
@TL(15)
(**************************************** WARNING ********************************************
 *** The KEBA Kemro K2 System including software is not intended for safety control tasks! ***
 ***                       For further information see Comment tab!                        ***
 *********************************************************************************************)

IF di_SequenceInterruption THEN
   IF sv_bSequenceInterruption THEN
      evSequenceInterruptData.SequenceInterrupt := nSequenceContinue;
   ELSE
      evSequenceInterruptData.SequenceInterrupt := nSequenceInterrupt;
   END_IF;

   SET_EVENT(evSequenceInterrupt, evSequenceInterruptData);
END_IF;

@END_Body

@@@BEG_Comment@@@
@TL(0)

@@@END_Comment@@@

@BEG_Body
@TL(27)
(**************************************** WARNING ********************************************
 *** The KEBA Kemro K2 System including software is not intended for safety control tasks! ***
 ***                       For further information see Comment tab!                        ***
 *********************************************************************************************)

IF (sv_OperationMode = nSetup) OR (sv_OperationMode = nManual) THEN
   RETURN;
END_IF;

IF evSequInterruptData.SequenceInterrupt = nSequenceInterrupt THEN
   sv_bSequenceInterruption := TRUE;
   mbResetInterrupt := FALSE;

   //set led attribute to "flashing" during sequence interrupt
   sv_bLedHalfAutomatic_ledAttr := 16#3;
   sv_bLedFullAutomatic_ledAttr := 16#3;

   sv_bHMILedHalfAutomatic_ledAttr := sv_bLedHalfAutomatic_ledAttr;
   sv_bHMILedFullAutomatic_ledAttr := sv_bLedFullAutomatic_ledAttr;

   START_PROCESS_ALGORITHM(paSequenceInterrupted);
ELSE
   mbResetInterrupt := TRUE;
END_IF;

@END_Body

@@@BEG_Comment@@@
@TL(0)

@@@END_Comment@@@

@BEG_SfcBody
10 8 9

@BEG_SfcData 2
@StepSeq @RT(4)sseq @F 3
@Step @RT(6)S_Init @F @T @F @F @RT(0) @F
@AcbCont @RT(7)unnamed @F 1
@Acb @RT(7)Action9 @F @T @RT(1)P @RT(0) @F @F @T @TL(4)

mbLedHalfAutomaticAttrLinked := IS_LINKED(sv_bLedHalfAutomatic_ledAttr);
mbLedFullAutomaticAttrLinked := IS_LINKED(sv_bLedFullAutomatic_ledAttr);

@F

@Trans @RT(6)Trans1 @F @T @F @F @T @F @TL(2)
TRUE

@RT(6)Trans1 @F
@Loop @RT(4)loop @F 2
@StepSeq @RT(3)seq @F 3
@Step @RT(13)S_Interrupted @F @F @F @F @RT(0) @F
@AcbCont @RT(7)unnamed @F 0

@AltBranch @RT(3)alt @F 2
@TransSeq @RT(4)tseq @F 3
@Trans @RT(15)TResetInterrupt @F @T @F @F @T @F @TL(2)
mbResetInterrupt

@RT(6)Trans2 @F
@Step @RT(12)S_WaitNoMove @F @F @F @F @RT(0) @F
@AcbCont @RT(7)unnamed @F 0

@Trans @RT(17)TNoMovementActive @F @T @F @F @T @F @TL(2)
sv_ActiveMovements.iNumberOfActiveMovements = 0

@RT(6)Trans4 @F

@TransSeq @RT(4)tseq @F 1
@Trans @RT(14)TOpModeChanged @F @T @T @F @T @F @TL(2)
sv_OperationMode < nHalfAutomatic

@RT(6)Trans8 @F

@Step @RT(6)S_Stop @F @F @F @F @RT(0) @F
@AcbCont @RT(7)unnamed @F 2
@Acb @RT(6)AReset @F @T @RT(1)P @RT(0) @F @F @T @TL(14)
sv_bSequenceInterruption := FALSE;
//set led attribute to "not flashing"
sv_bHMILedHalfAutomatic_ledAttr := 16#1;
sv_bHMILedFullAutomatic_ledAttr := 16#1;

IF mbLedHalfAutomaticAttrLinked THEN
   sv_bLedHalfAutomatic_ledAttr := sv_bHMILedHalfAutomatic_ledAttr;
END_IF;

IF mbLedFullAutomaticAttrLinked THEN
   sv_bLedFullAutomatic_ledAttr := sv_bHMILedFullAutomatic_ledAttr;
END_IF;

@F
@Acb @RT(5)AStop @F @T @RT(1)P @RT(0) @F @F @T @TL(2)
STOP_PROCESS_ALGORITHM();

@F

@Trans @RT(6)Trans3 @F @T @T @T @T @T @TL(2)
TRUE

@RT(6)Trans3 @F

@END_SfcData
@SaActions 1
@SaText @RT(7)Action9 1 @TL(0)

@SaTrans 0
@SaExits 0
@END_SfcBody

@@@BEG_Comment@@@
@TL(0)

@@@END_Comment@@@
@END_Body

@END_Contents

(* ---- ABShotCounter.pu ---- *)
(*
@h    ! WARNING !
@h    The Kemro K2 system (including software) only meets category B according to EN 954-1,
@h    thus it is not intended for usage in safety-relevant control applications in the field
@h    of personal safety (e.g. emergency stop).
@h    To implement potentially necessary safety-relevant control tasks, always use additional
@h    external safety devices that are intended for the particular purpose, and meet the necessary
@h    functional safety.
@h    For further information see EN 954-1 (EN ISO 13849-1) and/or the K2-x00 user manual, chapter
@h    "CE conformity, directives and standards".

Folowing functions are implemented in this block
- reset shot counter (by hmi or after loading mold data)
- maintenance of production counter
- stop cycle if set production counter is reached
- register movement for increasing shot counter

@FunctionID: S_ALLG_13
*)

IMPORT_OVER_LISTFILE
 SET_ALARM
, tnDataState
, tsMoveData
, tevStart
, tsDeviceId
, ABProduction
, ABMovementRegister
, tevStartData

END_IMPORT

ALGORITHM_BLOCK ABShotCounter #DUMMY_EDIT_BLOCK

SYSTEM_VAR
 sv_bResetShotCounter : BOOL;
 sv_iProdCounterAct : DINT;
 sv_iCavities : DINT;
 sv_iProdCounterSet : DINT (* shot limit *);
 sv_bTIGAvailable : BOOL;
 sv_iShotCounterAct : DINT;
 sv_bUseProdCounter : BOOL (* use shot counter *);
 sv_DataState : tnDataState;
 sv_bInitStart : BOOL;
 sv_MoveShotCounter : tsMoveData;
 sv_DeviceId : tsDeviceId;
 sv_iShotCounterRetain : UDINT;
 sv_rProdTimeAct : REAL;
 sv_rProdTimeTotal : REAL;
 sv_rProdTimeRemaining : REAL;
 sv_iProdCounterRemaining : DINT;
 sv_dCycleTime : TIME;
 sv_dLastCycleTime : TIME;
 sv_bEvenCycle : BOOL;
 sv_dCycleDelaySet : TIME;
 sv_iProdStartCounter : DINT;
 sv_sMoldData : STRING(99);
END_VAR

SYSTEM_OBJECT
 PU_Task_7 : TASK;
 erProdLimitReached : ALARM;
 TaskSlow : TASK;
 EV_Task_3 : TASK;
 evStart : tevStart;
END_OBJECT

VAR
 mbTIGAvailable : BOOL;
 abProduction : ABProduction;
END_VAR

(*
Calculates the productiontimes depending on the productcounter and cavities
*)

ALGORITHM aCalcProdTimes

VAR_INPUT
 dCycleTime : TIME (* cycle time, which should be used for calculation *);
END_VAR

VAR
 iRemainingShots : DINT;
END_VAR
#BEGIN_EDIT_BLOCK
(**************************************** WARNING ********************************************
 *** The KEBA Kemro K2 System including software is not intended for safety control tasks! ***
 ***                       For further information see Comment tab!                        ***
 *********************************************************************************************)

//Calculates the remaining production time in hours
IF (sv_iProdCounterAct <= sv_iProdCounterSet) THEN

   sv_iProdCounterRemaining := sv_iProdCounterSet - sv_iProdCounterAct;

   //calculate remaining shots (consider number of cavities!)
   iRemainingShots := (sv_iProdCounterRemaining / sv_iCavities);
   IF MOD(sv_iProdCounterRemaining, sv_iCavities) <> 0 THEN
      iRemainingShots := iRemainingShots + 1;
   END_IF;

   sv_rProdTimeRemaining := DINT_TO_REAL(iRemainingShots) * (LINT_TO_REAL(TIME_TO_LINT(dCycleTime))/1000000.0/3600.0);
   sv_rProdTimeTotal := sv_rProdTimeAct + sv_rProdTimeRemaining;

ELSE
   sv_rProdTimeRemaining := 0.0;
   sv_iProdCounterRemaining := 0;
END_IF;

;#END_EDIT_BLOCK END_ALGORITHM

POSTUPDATE_ALGORITHM pReCalcProdTimes ON PU_Task_7 WITH sv_iProdCounterSet,sv_iCavities

#BEGIN_EDIT_BLOCK
(**************************************** WARNING ********************************************
 *** The KEBA Kemro K2 System including software is not intended for safety control tasks! ***
 ***                       For further information see Comment tab!                        ***
 *********************************************************************************************)

//use last cycle time because the production counter can be changed
//during a running autocycle (sv_dCycleTime is not correct in this situation)
//sv_dLastCycleTime already includes cycle delay time
aCalcProdTimes(dCycleTime := sv_dLastCycleTime);

;#END_EDIT_BLOCK END_ALGORITHM

POSTUPDATE_ALGORITHM pResetShotCounter ON PU_Task_7 WITH sv_bResetShotCounter

#BEGIN_EDIT_BLOCK
(**************************************** WARNING ********************************************
 *** The KEBA Kemro K2 System including software is not intended for safety control tasks! ***
 ***                       For further information see Comment tab!                        ***
 *********************************************************************************************)

IF sv_bResetShotCounter THEN
    //reset shot counter
    sv_iShotCounterAct := 0;
    sv_iProdCounterAct := 0;
    abProduction.aResetData();
    sv_bResetShotCounter := FALSE;
    sv_rProdTimeAct := 0.0;
    sv_rProdTimeRemaining := 0.0;
    sv_rProdTimeTotal := 0.0;
    sv_iProdCounterRemaining := 0;
    sv_iProdStartCounter := sv_iProdStartCounter + 1;
END_IF;

;#END_EDIT_BLOCK END_ALGORITHM

POSTUPDATE_ALGORITHM pLoadSaveMoldData ON PU_Task_7 WITH sv_DataState

VAR
 bLoadMoldDataInProgress : BOOL;
 bSaveMoldDataInProgress : BOOL;
 sMoldData : STRING(99);
END_VAR
#BEGIN_EDIT_BLOCK
(**************************************** WARNING ********************************************
 *** The KEBA Kemro K2 System including software is not intended for safety control tasks! ***
 ***                       For further information see Comment tab!                        ***
 *********************************************************************************************)

IF (sv_DataState = nReadMoldData) THEN
    bLoadMoldDataInProgress := TRUE;
ELSIF (sv_DataState = nWriteMoldData) THEN
    bSaveMoldDataInProgress := TRUE;
    sMoldData := sv_sMoldData;
END_IF;

IF sv_DataState = nReady THEN
    //mold data loading/saving finished -> reset shot counter
    //mold data saving also indicates the start of a new production
    IF (bLoadMoldDataInProgress OR (bSaveMoldDataInProgress AND sMoldData <> sv_sMoldData)) THEN
        sv_bResetShotCounter := TRUE;
    END_IF;
    bSaveMoldDataInProgress := FALSE;
    bLoadMoldDataInProgress := FALSE;
END_IF;

;#END_EDIT_BLOCK END_ALGORITHM

PROCESS_ALGORITHM paInit ON TaskSlow AUTOSTART

#BEGIN_EDIT_BLOCK
(**************************************** WARNING ********************************************
 *** The KEBA Kemro K2 System including software is not intended for safety control tasks! ***
 ***                       For further information see Comment tab!                        ***
 *********************************************************************************************)

IF IS_LINKED(sv_bTIGAvailable) THEN
    mbTIGAvailable := sv_bTIGAvailable;
END_IF;

STOP_PROCESS_ALGORITHM();

;#END_EDIT_BLOCK END_ALGORITHM

POSTUPDATE_ALGORITHM pInitStart ON PU_Task_7 WITH sv_bInitStart

VAR
 abMoveShotCounterRegister : ABMovementRegister;
END_VAR
#BEGIN_EDIT_BLOCK
(**************************************** WARNING ********************************************
 *** The KEBA Kemro K2 System including software is not intended for safety control tasks! ***
 ***                       For further information see Comment tab!                        ***
 *********************************************************************************************)

IF sv_bInitStart THEN
   //register movement for shotcounter increasing
   abMoveShotCounterRegister.aRegister(@sv_MoveShotCounter);
END_IF;

sv_bEvenCycle := (MOD(sv_iShotCounterAct, 2) = 0);

;#END_EDIT_BLOCK END_ALGORITHM

ALGORITHM aCalcProdCnt

#BEGIN_EDIT_BLOCK
(**************************************** WARNING ********************************************
 *** The KEBA Kemro K2 System including software is not intended for safety control tasks! ***
 ***                       For further information see Comment tab!                        ***
 *********************************************************************************************)

IF NOT mbTIGAvailable THEN // calculate production counter here, if TIG available then production counter is set in FU TIG
   IF sv_iShotCounterAct <> 0 THEN
       sv_iProdCounterAct := sv_iProdCounterAct + sv_iCavities;
   END_IF;
END_IF;

// check production limit
IF (sv_iProdCounterAct >= sv_iProdCounterSet) AND sv_bUseProdCounter THEN
   SET_ALARM(Name := erProdLimitReached);
END_IF;

;#END_EDIT_BLOCK END_ALGORITHM

(*
taskslot is assigned to execute before evaFinishCycleAndStop in ABODC.pu
*)

EVENT_ALGORITHM evaStart ON EV_Task_3(100) WITH evStart

VAR_INPUT
 evStartData : tevStartData;
END_VAR
#BEGIN_EDIT_BLOCK
(**************************************** WARNING ********************************************
 *** The KEBA Kemro K2 System including software is not intended for safety control tasks! ***
 ***                       For further information see Comment tab!                        ***
 *********************************************************************************************)

IF evStartData.DeviceId <> sv_DeviceId THEN
   RETURN;
END_IF;

IF evStartData.MoveDir = sv_MoveShotCounter.MoveDir AND evStartData.MoveId = sv_MoveShotCounter.MoveId THEN

   //increase shot counter
   abProduction.aNewCycle();
   sv_iShotCounterRetain := sv_iShotCounterRetain + 1;

   sv_iShotCounterAct := sv_iShotCounterAct + 1;
   sv_rProdTimeAct := sv_rProdTimeAct + (LINT_TO_REAL(TIME_TO_LINT(sv_dCycleTime))/1000000.0/3600.0);

   sv_bEvenCycle := (MOD(sv_iShotCounterAct, 2) = 0);

   aCalcProdCnt();

   aCalcProdTimes(dCycleTime := (sv_dCycleTime + sv_dCycleDelaySet));
END_IF;

;#END_EDIT_BLOCK END_ALGORITHM

END_ALGORITHM_BLOCK

#END_OF_IEC_PART

@Puma @IecEditor 6 94 @Pou 25
@@@BEG_Comment@@@
@h    ! WARNING !
@h    The Kemro K2 system (including software) only meets category B according to EN 954-1,
@h    thus it is not intended for usage in safety-relevant control applications in the field
@h    of personal safety (e.g. emergency stop).
@h    To implement potentially necessary safety-relevant control tasks, always use additional
@h    external safety devices that are intended for the particular purpose, and meet the necessary
@h    functional safety.
@h    For further information see EN 954-1 (EN ISO 13849-1) and/or the K2-x00 user manual, chapter
@h    "CE conformity, directives and standards".

Folowing functions are implemented in this block
- reset shot counter (by hmi or after loading mold data)
- maintenance of production counter
- stop cycle if set production counter is reached
- register movement for increasing shot counter

@FunctionID: S_ALLG_13
@@@END_Comment@@@

@BEG_Contents

@BEG_Func
@RT(17)FuncTreeContainer
1
@Var @RT(9)SET_ALARM @RT(0) @T @T @DERIVED 0 @F @RT(23)KEBA_STANDARD_PROCEDURE @F
@T
@BEG_Attrib
0 @RT(0) @RT(0)
@END_Attrib
1 1 @F @F @F @F

@END_Func

@BEG_Const
@RT(18)ConstTreeContainer
0
@END_Const

@BEG_Export

@BEG_Kind
@ALGORITHM_BLOCK @RT(13)ABShotCounter @STRUCTURED_TEXT
@RT(0) @RT(0) @RT(0)
@END_Kind

@BEG_Dcl
@RT(16)DclTreeContainer
29
@Var @RT(9)PU_Task_7 @RT(0) @T @T @RENAMED 0 @T @T @DT @RT(4)TASK @RT(0) @T @T @BASIC 0 @F
@F @F
@T
@BEG_Attrib
3 @RT(0) @RT(0) @RT(0)
@END_Attrib
1 7 @F @F @F @F

@Var @RT(20)sv_bResetShotCounter @RT(0) @T @T @RENAMED 0 @T @T @DT @RT(4)BOOL @RT(0) @T @T @BASIC 0 @F
@F @F
@T
@BEG_Attrib
3 @RT(0) @RT(0) @RT(0)
@END_Attrib
1 8 @F @F @F @F

@Var @RT(18)sv_iProdCounterAct @RT(0) @T @F @DT @RT(4)DINT @RT(0) @T @T @BASIC 0 @F
@F @F
@T
@BEG_Attrib
3 @RT(0) @RT(0) @RT(0)
@END_Attrib
1 8 @F @F @F @F

@Var @RT(12)sv_iCavities @RT(0) @T @F @DT @RT(4)DINT @RT(0) @T @T @BASIC 0 @F
@F @F
@T
@BEG_Attrib
3 @RT(0) @RT(0) @RT(0)
@END_Attrib
1 8 @F @F @F @F

@Var @RT(18)sv_iProdCounterSet @RT(0) @T @F @DT @RT(4)DINT @RT(0) @T @T @BASIC 0 @F
@F @F
@T
@BEG_Attrib
3 @RT(0) @RT(10)shot limit @RT(0)
@END_Attrib
1 8 @F @F @F @F

@Var @RT(18)erProdLimitReached @RT(0) @T @F @DT @RT(5)ALARM @RT(0) @T @T @BASIC 0 @F
@F @F
@T
@BEG_Attrib
3 @RT(0) @RT(0) @RT(0)
@END_Attrib
1 7 @F @F @F @F

@Var @RT(16)sv_bTIGAvailable @RT(0) @T @F @DT @RT(4)BOOL @RT(0) @T @T @BASIC 0 @F
@F @F
@T
@BEG_Attrib
3 @RT(0) @RT(0) @RT(0)
@END_Attrib
1 8 @F @F @F @F

@Var @RT(18)sv_iShotCounterAct @RT(0) @T @F @DT @RT(4)DINT @RT(0) @T @T @BASIC 0 @F
@F @F
@T
@BEG_Attrib
3 @RT(0) @RT(0) @RT(0)
@END_Attrib
1 8 @F @F @F @F

@Var @RT(18)sv_bUseProdCounter @RT(0) @T @F @DT @RT(4)BOOL @RT(0) @T @T @BASIC 0 @F
@F @F
@T
@BEG_Attrib
3 @RT(0) @RT(16)use shot counter @RT(0)
@END_Attrib
1 8 @F @F @F @F

@Var @RT(12)sv_DataState @RT(0) @T @T @DERIVED 0 @T @T @DT @RT(11)tnDataState @RT(0) @T @T @UNKNOWN 0 @F
@F @F
@T
@BEG_Attrib
3 @RT(0) @RT(0) @RT(0)
@END_Attrib
1 8 @F @F @F @F

@Var @RT(8)TaskSlow @RT(0) @T @F @DT @RT(4)TASK @RT(0) @T @T @BASIC 0 @F
@F @F
@T
@BEG_Attrib
3 @RT(0) @RT(0) @RT(0)
@END_Attrib
1 7 @F @F @F @F

@Var @RT(14)mbTIGAvailable @RT(0) @T @F @DT @RT(4)BOOL @RT(0) @T @T @BASIC 0 @F
@F @F
@T
@BEG_Attrib
3 @RT(0) @RT(0) @RT(0)
@END_Attrib
1 0 @F @F @F @F

@Var @RT(13)sv_bInitStart @RT(0) @T @F @DT @RT(4)BOOL @RT(0) @T @T @BASIC 0 @F
@F @F
@T
@BEG_Attrib
3 @RT(0) @RT(0) @RT(0)
@END_Attrib
1 8 @F @F @F @F

@Var @RT(18)sv_MoveShotCounter @RT(0) @T @T @DERIVED 0 @T @T @DT @RT(10)tsMoveData @RT(0) @T @T @UNKNOWN 0 @F
@F @F
@T
@BEG_Attrib
3 @RT(0) @RT(0) @RT(0)
@END_Attrib
1 8 @F @F @F @F

@Var @RT(9)EV_Task_3 @RT(0) @T @F @DT @RT(4)TASK @RT(0) @T @T @BASIC 0 @F
@F @F
@T
@BEG_Attrib
3 @RT(0) @RT(0) @RT(0)
@END_Attrib
1 7 @F @F @F @F

@Var @RT(7)evStart @RT(0) @T @T @DERIVED 0 @T @T @DT @RT(8)tevStart @RT(0) @T @T @UNKNOWN 0 @F
@F @F
@T
@BEG_Attrib
3 @RT(0) @RT(0) @RT(0)
@END_Attrib
1 7 @F @F @F @F

@Var @RT(11)sv_DeviceId @RT(0) @T @T @DERIVED 0 @T @T @DT @RT(10)tsDeviceId @RT(0) @T @T @UNKNOWN 0 @F
@F @F
@T
@BEG_Attrib
3 @RT(0) @RT(0) @RT(0)
@END_Attrib
1 8 @F @F @F @F

@Var @RT(21)sv_iShotCounterRetain @RT(0) @T @F @DT @RT(5)UDINT @RT(0) @T @T @BASIC 0 @F
@F @F
@T
@BEG_Attrib
3 @RT(0) @RT(0) @RT(0)
@END_Attrib
1 8 @F @F @F @F

@Var @RT(12)abProduction @RT(0) @T @T @DERIVED 0 @T @T @DT @RT(12)ABProduction @RT(0) @T @T @UNKNOWN 0 @F
@F @F
@T
@BEG_Attrib
3 @RT(0) @RT(0) @RT(0)
@END_Attrib
1 0 @F @F @F @F

@Var @RT(15)sv_rProdTimeAct @RT(0) @T @F @DT @RT(4)REAL @RT(0) @T @T @BASIC 0 @F
@F @F
@T
@BEG_Attrib
3 @RT(0) @RT(0) @RT(0)
@END_Attrib
1 8 @F @F @F @F

@Var @RT(17)sv_rProdTimeTotal @RT(0) @T @F @DT @RT(4)REAL @RT(0) @T @T @BASIC 0 @F
@F @F
@T
@BEG_Attrib
3 @RT(0) @RT(0) @RT(0)
@END_Attrib
1 8 @F @F @F @F

@Var @RT(21)sv_rProdTimeRemaining @RT(0) @T @F @DT @RT(4)REAL @RT(0) @T @T @BASIC 0 @F
@F @F
@T
@BEG_Attrib
3 @RT(0) @RT(0) @RT(0)
@END_Attrib
1 8 @F @F @F @F

@Var @RT(24)sv_iProdCounterRemaining @RT(0) @T @F @DT @RT(4)DINT @RT(0) @T @T @BASIC 0 @F
@F @F
@T
@BEG_Attrib
3 @RT(0) @RT(0) @RT(0)
@END_Attrib
1 8 @F @F @F @F

@Var @RT(13)sv_dCycleTime @RT(0) @T @F @DT @RT(4)TIME @RT(0) @T @T @BASIC 0 @F
@F @F
@T
@BEG_Attrib
3 @RT(0) @RT(0) @RT(0)
@END_Attrib
1 8 @F @F @F @F

@Var @RT(17)sv_dLastCycleTime @RT(0) @T @F @DT @RT(4)TIME @RT(0) @T @T @BASIC 0 @F
@F @F
@T
@BEG_Attrib
3 @RT(0) @RT(0) @RT(0)
@END_Attrib
1 8 @F @F @F @F

@Var @RT(13)sv_bEvenCycle @RT(0) @T @F @DT @RT(4)BOOL @RT(0) @T @T @BASIC 0 @F
@F @F
@T
@BEG_Attrib
3 @RT(0) @RT(0) @RT(0)
@END_Attrib
1 8 @F @F @F @F

@Var @RT(17)sv_dCycleDelaySet @RT(0) @T @F @DT @RT(4)TIME @RT(0) @T @T @BASIC 0 @F
@F @F
@T
@BEG_Attrib
3 @RT(0) @RT(0) @RT(0)
@END_Attrib
1 8 @F @F @F @F

@Var @RT(20)sv_iProdStartCounter @RT(0) @T @F @DT @RT(4)DINT @RT(0) @T @T @BASIC 0 @F
@F @F
@T
@BEG_Attrib
3 @RT(0) @RT(0) @RT(0)
@END_Attrib
1 8 @F @F @F @F

@Var @RT(12)sv_sMoldData @RT(0) @T @F @DT @RT(10)STRING(99) @RT(0) @T @T @STRING 0 @F @RT(2)99 @F
@F @F
@T
@BEG_Attrib
3 @RT(0) @RT(0) @RT(0)
@END_Attrib
1 8 @F @F @F @F

@END_Dcl

@END_Export

@BEG_Body

8

@BEG_Export

@BEG_Algo
@ALGORITHM @RT(14)aCalcProdTimes @STRUCTURED_TEXT
@RT(0) @RT(0) @RT(0) @F @F
@END_Algo

@BEG_Dcl
@RT(16)DclTreeContainer
2
@Var @RT(10)dCycleTime @RT(0) @T @F @DT @RT(4)TIME @RT(0) @T @T @BASIC 0 @F
@F @F
@T
@BEG_Attrib
3 @RT(0) @RT(48)cycle time, which should be used for calculation @RT(0)
@END_Attrib
1 1 @F @F @F @F

@Var @RT(15)iRemainingShots @RT(0) @T @F @DT @RT(4)DINT @RT(0) @T @T @BASIC 0 @F
@F @F
@T
@BEG_Attrib
3 @RT(0) @RT(0) @RT(0)
@END_Attrib
1 0 @F @F @F @F

@END_Dcl

@END_Export

@BEG_Export

@BEG_Algo
@POSTUPDATE_ALGORITHM @RT(16)pReCalcProdTimes @STRUCTURED_TEXT
@RT(0) @RT(31)sv_iProdCounterSet,sv_iCavities @RT(9)PU_Task_7 @F @F
@END_Algo

@BEG_Dcl
@RT(16)DclTreeContainer
0
@END_Dcl

@END_Export

@BEG_Export

@BEG_Algo
@POSTUPDATE_ALGORITHM @RT(17)pResetShotCounter @STRUCTURED_TEXT
@RT(0) @RT(20)sv_bResetShotCounter @RT(9)PU_Task_7 @F @F
@END_Algo

@BEG_Dcl
@RT(16)DclTreeContainer
0
@END_Dcl

@END_Export

@BEG_Export

@BEG_Algo
@POSTUPDATE_ALGORITHM @RT(17)pLoadSaveMoldData @STRUCTURED_TEXT
@RT(0) @RT(12)sv_DataState @RT(9)PU_Task_7 @F @F
@END_Algo

@BEG_Dcl
@RT(16)DclTreeContainer
3
@Var @RT(23)bLoadMoldDataInProgress @RT(0) @T @F @DT @RT(4)BOOL @RT(0) @T @T @BASIC 0 @F
@F @F
@T
@BEG_Attrib
3 @RT(0) @RT(0) @RT(0)
@END_Attrib
1 0 @F @F @F @F

@Var @RT(23)bSaveMoldDataInProgress @RT(0) @T @F @DT @RT(4)BOOL @RT(0) @T @T @BASIC 0 @F
@F @F
@T
@BEG_Attrib
3 @RT(0) @RT(0) @RT(0)
@END_Attrib
1 0 @F @F @F @F

@Var @RT(9)sMoldData @RT(0) @T @F @DT @RT(10)STRING(99) @RT(0) @T @T @STRING 0 @F @RT(2)99 @F
@F @F
@T
@BEG_Attrib
3 @RT(0) @RT(0) @RT(0)
@END_Attrib
1 0 @F @F @F @F

@END_Dcl

@END_Export

@BEG_Export

@BEG_Algo
@PROCESS_ALGORITHM @RT(6)paInit @STRUCTURED_TEXT
@RT(0) @RT(0) @RT(8)TaskSlow @T @F
@END_Algo

@BEG_Dcl
@RT(16)DclTreeContainer
0
@END_Dcl

@END_Export

@BEG_Export

@BEG_Algo
@POSTUPDATE_ALGORITHM @RT(10)pInitStart @STRUCTURED_TEXT
@RT(0) @RT(13)sv_bInitStart @RT(9)PU_Task_7 @F @F
@END_Algo

@BEG_Dcl
@RT(16)DclTreeContainer
1
@Var @RT(25)abMoveShotCounterRegister @RT(0) @T @T @DERIVED 0 @T @T @DT @RT(18)ABMovementRegister @RT(0) @T @T @UNKNOWN 0 @F
@F @F
@T
@BEG_Attrib
3 @RT(0) @RT(0) @RT(0)
@END_Attrib
1 0 @F @F @F @F

@END_Dcl

@END_Export

@BEG_Export

@BEG_Algo
@ALGORITHM @RT(12)aCalcProdCnt @STRUCTURED_TEXT
@RT(0) @RT(0) @RT(0) @F @F
@END_Algo

@BEG_Dcl
@RT(16)DclTreeContainer
0
@END_Dcl

@END_Export

@BEG_Export

@BEG_Algo
@EVENT_ALGORITHM @RT(8)evaStart @STRUCTURED_TEXT
@RT(0) @RT(7)evStart @RT(14)EV_Task_3(100) @F @F
@END_Algo

@BEG_Dcl
@RT(16)DclTreeContainer
1
@Var @RT(11)evStartData @RT(0) @T @T @DERIVED 0 @T @T @DT @RT(12)tevStartData @RT(0) @T @T @UNKNOWN 0 @F
@F @F
@T
@BEG_Attrib
3 @RT(0) @RT(0) @RT(0)
@END_Attrib
1 1 @F @F @F @F

@END_Dcl

@END_Export

@BEG_Body
@TL(24)
(**************************************** WARNING ********************************************
 *** The KEBA Kemro K2 System including software is not intended for safety control tasks! ***
 ***                       For further information see Comment tab!                        ***
 *********************************************************************************************)

//Calculates the remaining production time in hours
IF (sv_iProdCounterAct <= sv_iProdCounterSet) THEN

   sv_iProdCounterRemaining := sv_iProdCounterSet - sv_iProdCounterAct;

   //calculate remaining shots (consider number of cavities!)
   iRemainingShots := (sv_iProdCounterRemaining / sv_iCavities);
   IF MOD(sv_iProdCounterRemaining, sv_iCavities) <> 0 THEN
      iRemainingShots := iRemainingShots + 1;
   END_IF;

   sv_rProdTimeRemaining := DINT_TO_REAL(iRemainingShots) * (LINT_TO_REAL(TIME_TO_LINT(dCycleTime))/1000000.0/3600.0);
   sv_rProdTimeTotal := sv_rProdTimeAct + sv_rProdTimeRemaining;

ELSE
   sv_rProdTimeRemaining := 0.0;
   sv_iProdCounterRemaining := 0;
END_IF;

@END_Body

@@@BEG_Comment@@@
@TL(1)
Calculates the productiontimes depending on the productcounter and cavities
@@@END_Comment@@@

@BEG_Body
@TL(10)
(**************************************** WARNING ********************************************
 *** The KEBA Kemro K2 System including software is not intended for safety control tasks! ***
 ***                       For further information see Comment tab!                        ***
 *********************************************************************************************)

//use last cycle time because the production counter can be changed
//during a running autocycle (sv_dCycleTime is not correct in this situation)
//sv_dLastCycleTime already includes cycle delay time
aCalcProdTimes(dCycleTime := sv_dLastCycleTime);

@END_Body

@@@BEG_Comment@@@
@TL(0)

@@@END_Comment@@@

@BEG_Body
@TL(18)
(**************************************** WARNING ********************************************
 *** The KEBA Kemro K2 System including software is not intended for safety control tasks! ***
 ***                       For further information see Comment tab!                        ***
 *********************************************************************************************)

IF sv_bResetShotCounter THEN
    //reset shot counter
    sv_iShotCounterAct := 0;
    sv_iProdCounterAct := 0;
    abProduction.aResetData();
    sv_bResetShotCounter := FALSE;
    sv_rProdTimeAct := 0.0;
    sv_rProdTimeRemaining := 0.0;
    sv_rProdTimeTotal := 0.0;
    sv_iProdCounterRemaining := 0;
    sv_iProdStartCounter := sv_iProdStartCounter + 1;
END_IF;

@END_Body

@@@BEG_Comment@@@
@TL(0)

@@@END_Comment@@@

@BEG_Body
@TL(22)
(**************************************** WARNING ********************************************
 *** The KEBA Kemro K2 System including software is not intended for safety control tasks! ***
 ***                       For further information see Comment tab!                        ***
 *********************************************************************************************)

IF (sv_DataState = nReadMoldData) THEN
    bLoadMoldDataInProgress := TRUE;
ELSIF (sv_DataState = nWriteMoldData) THEN
    bSaveMoldDataInProgress := TRUE;
    sMoldData := sv_sMoldData;
END_IF;

IF sv_DataState = nReady THEN
    //mold data loading/saving finished -> reset shot counter
    //mold data saving also indicates the start of a new production
    IF (bLoadMoldDataInProgress OR (bSaveMoldDataInProgress AND sMoldData <> sv_sMoldData)) THEN
        sv_bResetShotCounter := TRUE;
    END_IF;
    bSaveMoldDataInProgress := FALSE;
    bLoadMoldDataInProgress := FALSE;
END_IF;

@END_Body

@@@BEG_Comment@@@
@TL(0)

@@@END_Comment@@@

@BEG_Body
@TL(11)
(**************************************** WARNING ********************************************
 *** The KEBA Kemro K2 System including software is not intended for safety control tasks! ***
 ***                       For further information see Comment tab!                        ***
 *********************************************************************************************)

IF IS_LINKED(sv_bTIGAvailable) THEN
    mbTIGAvailable := sv_bTIGAvailable;
END_IF;

STOP_PROCESS_ALGORITHM();

@END_Body

@@@BEG_Comment@@@
@TL(0)

@@@END_Comment@@@

@BEG_Body
@TL(13)
(**************************************** WARNING ********************************************
 *** The KEBA Kemro K2 System including software is not intended for safety control tasks! ***
 ***                       For further information see Comment tab!                        ***
 *********************************************************************************************)

IF sv_bInitStart THEN
   //register movement for shotcounter increasing
   abMoveShotCounterRegister.aRegister(@sv_MoveShotCounter);
END_IF;

sv_bEvenCycle := (MOD(sv_iShotCounterAct, 2) = 0);

@END_Body

@@@BEG_Comment@@@
@TL(0)

@@@END_Comment@@@

@BEG_Body
@TL(16)
(**************************************** WARNING ********************************************
 *** The KEBA Kemro K2 System including software is not intended for safety control tasks! ***
 ***                       For further information see Comment tab!                        ***
 *********************************************************************************************)

IF NOT mbTIGAvailable THEN // calculate production counter here, if TIG available then production counter is set in FU TIG
   IF sv_iShotCounterAct <> 0 THEN
       sv_iProdCounterAct := sv_iProdCounterAct + sv_iCavities;
   END_IF;
END_IF;

// check production limit
IF (sv_iProdCounterAct >= sv_iProdCounterSet) AND sv_bUseProdCounter THEN
   SET_ALARM(Name := erProdLimitReached);
END_IF;

@END_Body

@@@BEG_Comment@@@
@TL(0)

@@@END_Comment@@@

@BEG_Body
@TL(25)
(**************************************** WARNING ********************************************
 *** The KEBA Kemro K2 System including software is not intended for safety control tasks! ***
 ***                       For further information see Comment tab!                        ***
 *********************************************************************************************)

IF evStartData.DeviceId <> sv_DeviceId THEN
   RETURN;
END_IF;

IF evStartData.MoveDir = sv_MoveShotCounter.MoveDir AND evStartData.MoveId = sv_MoveShotCounter.MoveId THEN

   //increase shot counter
   abProduction.aNewCycle();
   sv_iShotCounterRetain := sv_iShotCounterRetain + 1;

   sv_iShotCounterAct := sv_iShotCounterAct + 1;
   sv_rProdTimeAct := sv_rProdTimeAct + (LINT_TO_REAL(TIME_TO_LINT(sv_dCycleTime))/1000000.0/3600.0);

   sv_bEvenCycle := (MOD(sv_iShotCounterAct, 2) = 0);

   aCalcProdCnt();

   aCalcProdTimes(dCycleTime := (sv_dCycleTime + sv_dCycleDelaySet));
END_IF;

@END_Body

@@@BEG_Comment@@@
@TL(1)
taskslot is assigned to execute before evaFinishCycleAndStop in ABODC.pu
@@@END_Comment@@@
@END_Body

@END_Contents

(* ---- ABSignalSetReset.pu ---- *)
IMPORT_OVER_LISTFILE
 ABAlarmSignalList
, ALARM_EVENT
, ALARM_EVENT_DATA
, tsElementAlarmSignal

END_IMPORT

ALGORITHM_BLOCK ABSignalSetReset #DUMMY_EDIT_BLOCK

SYSTEM_VAR
 sv_bSetAlarmSignal : BOOL;
 sv_iSetAlarmSignalCount : DINT (* counter how many alarms requested the alarm signal (incremented with evAlarmLampBlink event; decremented with evAlarmLampReset) *);
END_VAR

SYSTEM_OBJECT
 evAlarmLampBlink : ALARM_EVENT;
 evAlarmLampReset : ALARM_EVENT;
 EV_Task_3 : TASK;
END_OBJECT

VAR
 abAlarmSignalList : ABAlarmSignalList;
 mbInitDone : BOOL;
END_VAR

EVENT_ALGORITHM evaAlarmLampBlink ON EV_Task_3 WITH evAlarmLampBlink

VAR_INPUT
 evAlarmAlarmSignalData : ALARM_EVENT_DATA;
END_VAR

VAR
 ElementAlarmSignal : tsElementAlarmSignal;
END_VAR
#BEGIN_EDIT_BLOCK
IF NOT mbInitDone THEN
    abAlarmSignalList.aInit();
    mbInitDone := TRUE;
END_IF;

//search if entry already exists
ElementAlarmSignal.SearchData.Alarm := evAlarmAlarmSignalData.NAME;
ElementAlarmSignal.SearchData.SubID1 := evAlarmAlarmSignalData.SUBID1;
ElementAlarmSignal.SearchData.SubID2 := evAlarmAlarmSignalData.SUBID2;
ElementAlarmSignal.SearchData.SubID3 := evAlarmAlarmSignalData.SUBID3;
ElementAlarmSignal.SearchData.SubID4 := evAlarmAlarmSignalData.SUBID4;

abAlarmSignalList.aSearch(SearchData := ElementAlarmSignal.SearchData);

IF NOT abAlarmSignalList.aSearch.bFound THEN
    //add entry
    ElementAlarmSignal.ElementData.Alarm := evAlarmAlarmSignalData.NAME;
    ElementAlarmSignal.ElementData.SubID1 := evAlarmAlarmSignalData.SUBID1;
    ElementAlarmSignal.ElementData.SubID2 := evAlarmAlarmSignalData.SUBID2;
    ElementAlarmSignal.ElementData.SubID3 := evAlarmAlarmSignalData.SUBID3;
    ElementAlarmSignal.ElementData.SubID4 := evAlarmAlarmSignalData.SUBID4;
    abAlarmSignalList.aAdd(Element := ElementAlarmSignal);
END_IF;

//get number of elements
sv_iSetAlarmSignalCount := abAlarmSignalList.aGetElementCount();
IF sv_iSetAlarmSignalCount > 0 THEN
    //one or more entries in the list -> set alarm signal
    sv_bSetAlarmSignal := TRUE;
END_IF;

;#END_EDIT_BLOCK END_ALGORITHM

EVENT_ALGORITHM evaAlarmLampReset ON EV_Task_3 WITH evAlarmLampReset

VAR_INPUT
 evAlarmMotorReleaseData : ALARM_EVENT_DATA;
END_VAR

VAR
 ElementMotorRelease : tsElementAlarmSignal;
END_VAR
#BEGIN_EDIT_BLOCK
IF NOT mbInitDone THEN
    abAlarmSignalList.aInit();
    mbInitDone := TRUE;
END_IF;

//search if entry already exists
ElementMotorRelease.SearchData.Alarm := evAlarmMotorReleaseData.NAME;
ElementMotorRelease.SearchData.SubID1 := evAlarmMotorReleaseData.SUBID1;
ElementMotorRelease.SearchData.SubID2 := evAlarmMotorReleaseData.SUBID2;
ElementMotorRelease.SearchData.SubID3 := evAlarmMotorReleaseData.SUBID3;
ElementMotorRelease.SearchData.SubID4 := evAlarmMotorReleaseData.SUBID4;

abAlarmSignalList.aSearch(SearchData := ElementMotorRelease.SearchData);

IF abAlarmSignalList.aSearch.bFound THEN
    //remove entry
    abAlarmSignalList.aRemove(SearchData := ElementMotorRelease.SearchData);
END_IF;

//get number of elements
sv_iSetAlarmSignalCount := abAlarmSignalList.aGetElementCount();
IF sv_iSetAlarmSignalCount = 0 THEN
    //no entries left -> reset alarm signal
    sv_bSetAlarmSignal := FALSE;
END_IF;

;#END_EDIT_BLOCK END_ALGORITHM

END_ALGORITHM_BLOCK

#END_OF_IEC_PART

@Puma @IecEditor 6 68 @Pou 25
@@@BEG_Comment@@@

@@@END_Comment@@@

@BEG_Contents

@BEG_Func
@RT(17)FuncTreeContainer
0
@END_Func

@BEG_Const
@RT(18)ConstTreeContainer
0
@END_Const

@BEG_Export

@BEG_Kind
@ALGORITHM_BLOCK @RT(16)ABSignalSetReset @STRUCTURED_TEXT
@RT(0) @RT(0) @RT(0)
@END_Kind

@BEG_Dcl
@RT(16)DclTreeContainer
7
@Var @RT(17)abAlarmSignalList @RT(0) @T @T @DERIVED 0 @T @T @DT @RT(17)ABAlarmSignalList @RT(0) @T @T @UNKNOWN 0 @F
@F @F
@T
@BEG_Attrib
3 @RT(0) @RT(0) @RT(0)
@END_Attrib
1 0 @F @F @F @F

@Var @RT(16)evAlarmLampBlink @RT(0) @T @T @RENAMED 0 @T @T @DT @RT(11)ALARM_EVENT @RT(0) @T @T @UNKNOWN 0 @F
@F @F
@T
@BEG_Attrib
3 @RT(0) @RT(0) @RT(0)
@END_Attrib
1 7 @F @F @F @F

@Var @RT(16)evAlarmLampReset @RT(0) @T @T @RENAMED 0 @T @T @DT @RT(11)ALARM_EVENT @RT(0) @T @T @UNKNOWN 0 @F
@F @F
@T
@BEG_Attrib
3 @RT(0) @RT(0) @RT(0)
@END_Attrib
1 7 @F @F @F @F

@Var @RT(9)EV_Task_3 @RT(0) @T @T @RENAMED 0 @T @T @DT @RT(4)TASK @RT(0) @T @T @BASIC 0 @F
@F @F
@T
@BEG_Attrib
3 @RT(0) @RT(0) @RT(0)
@END_Attrib
1 7 @F @F @F @F

@Var @RT(10)mbInitDone @RT(0) @T @F @DT @RT(4)BOOL @RT(0) @T @T @BASIC 0 @F
@F @F
@T
@BEG_Attrib
3 @RT(0) @RT(0) @RT(0)
@END_Attrib
1 0 @F @F @F @F

@Var @RT(18)sv_bSetAlarmSignal @RT(0) @T @F @DT @RT(4)BOOL @RT(0) @T @T @BASIC 0 @F
@F @F
@T
@BEG_Attrib
3 @RT(0) @RT(0) @RT(0)
@END_Attrib
1 8 @F @F @F @F

@Var @RT(23)sv_iSetAlarmSignalCount @RT(0) @T @F @DT @RT(4)DINT @RT(0) @T @T @BASIC 0 @F
@F @F
@T
@BEG_Attrib
3 @RT(0) @RT(127)counter how many alarms requested the alarm signal (incremented with evAlarmLampBlink event; decremented with evAlarmLampReset) @RT(0)
@END_Attrib
1 8 @F @F @F @F

@END_Dcl

@END_Export

@BEG_Body

2

@BEG_Export

@BEG_Algo
@EVENT_ALGORITHM @RT(17)evaAlarmLampBlink @STRUCTURED_TEXT
@RT(0) @RT(16)evAlarmLampBlink @RT(9)EV_Task_3 @F @F
@END_Algo

@BEG_Dcl
@RT(16)DclTreeContainer
2
@Var @RT(22)evAlarmAlarmSignalData @RT(0) @T @T @DERIVED 0 @T @T @DT @RT(16)ALARM_EVENT_DATA @RT(0) @T @T @UNKNOWN 0 @F
@F @F
@T
@BEG_Attrib
3 @RT(0) @RT(0) @RT(0)
@END_Attrib
1 1 @F @F @F @F

@Var @RT(18)ElementAlarmSignal @RT(0) @T @T @DERIVED 0 @T @T @DT @RT(20)tsElementAlarmSignal @RT(0) @T @T @UNKNOWN 0 @F
@F @F
@T
@BEG_Attrib
3 @RT(0) @RT(0) @RT(0)
@END_Attrib
1 0 @F @F @F @F

@END_Dcl

@END_Export

@BEG_Export

@BEG_Algo
@EVENT_ALGORITHM @RT(17)evaAlarmLampReset @STRUCTURED_TEXT
@RT(0) @RT(16)evAlarmLampReset @RT(9)EV_Task_3 @F @F
@END_Algo

@BEG_Dcl
@RT(16)DclTreeContainer
2
@Var @RT(23)evAlarmMotorReleaseData @RT(0) @T @T @DERIVED 0 @T @T @DT @RT(16)ALARM_EVENT_DATA @RT(0) @T @T @UNKNOWN 0 @F
@F @F
@T
@BEG_Attrib
3 @RT(0) @RT(0) @RT(0)
@END_Attrib
1 1 @F @F @F @F

@Var @RT(19)ElementMotorRelease @RT(0) @T @T @DERIVED 0 @T @T @DT @RT(20)tsElementAlarmSignal @RT(0) @T @T @UNKNOWN 0 @F
@F @F
@T
@BEG_Attrib
3 @RT(0) @RT(0) @RT(0)
@END_Attrib
1 0 @F @F @F @F

@END_Dcl

@END_Export

@BEG_Body
@TL(31)
IF NOT mbInitDone THEN
    abAlarmSignalList.aInit();
    mbInitDone := TRUE;
END_IF;

//search if entry already exists
ElementAlarmSignal.SearchData.Alarm := evAlarmAlarmSignalData.NAME;
ElementAlarmSignal.SearchData.SubID1 := evAlarmAlarmSignalData.SUBID1;
ElementAlarmSignal.SearchData.SubID2 := evAlarmAlarmSignalData.SUBID2;
ElementAlarmSignal.SearchData.SubID3 := evAlarmAlarmSignalData.SUBID3;
ElementAlarmSignal.SearchData.SubID4 := evAlarmAlarmSignalData.SUBID4;

abAlarmSignalList.aSearch(SearchData := ElementAlarmSignal.SearchData);

IF NOT abAlarmSignalList.aSearch.bFound THEN
    //add entry
    ElementAlarmSignal.ElementData.Alarm := evAlarmAlarmSignalData.NAME;
    ElementAlarmSignal.ElementData.SubID1 := evAlarmAlarmSignalData.SUBID1;
    ElementAlarmSignal.ElementData.SubID2 := evAlarmAlarmSignalData.SUBID2;
    ElementAlarmSignal.ElementData.SubID3 := evAlarmAlarmSignalData.SUBID3;
    ElementAlarmSignal.ElementData.SubID4 := evAlarmAlarmSignalData.SUBID4;
    abAlarmSignalList.aAdd(Element := ElementAlarmSignal);
END_IF;

//get number of elements
sv_iSetAlarmSignalCount := abAlarmSignalList.aGetElementCount();
IF sv_iSetAlarmSignalCount > 0 THEN
    //one or more entries in the list -> set alarm signal
    sv_bSetAlarmSignal := TRUE;
END_IF;

@END_Body

@@@BEG_Comment@@@
@TL(0)

@@@END_Comment@@@

@BEG_Body
@TL(26)
IF NOT mbInitDone THEN
    abAlarmSignalList.aInit();
    mbInitDone := TRUE;
END_IF;

//search if entry already exists
ElementMotorRelease.SearchData.Alarm := evAlarmMotorReleaseData.NAME;
ElementMotorRelease.SearchData.SubID1 := evAlarmMotorReleaseData.SUBID1;
ElementMotorRelease.SearchData.SubID2 := evAlarmMotorReleaseData.SUBID2;
ElementMotorRelease.SearchData.SubID3 := evAlarmMotorReleaseData.SUBID3;
ElementMotorRelease.SearchData.SubID4 := evAlarmMotorReleaseData.SUBID4;

abAlarmSignalList.aSearch(SearchData := ElementMotorRelease.SearchData);

IF abAlarmSignalList.aSearch.bFound THEN
    //remove entry
    abAlarmSignalList.aRemove(SearchData := ElementMotorRelease.SearchData);
END_IF;

//get number of elements
sv_iSetAlarmSignalCount := abAlarmSignalList.aGetElementCount();
IF sv_iSetAlarmSignalCount = 0 THEN
    //no entries left -> reset alarm signal
    sv_bSetAlarmSignal := FALSE;
END_IF;

@END_Body

@@@BEG_Comment@@@
@TL(0)

@@@END_Comment@@@
@END_Body

@END_Contents
